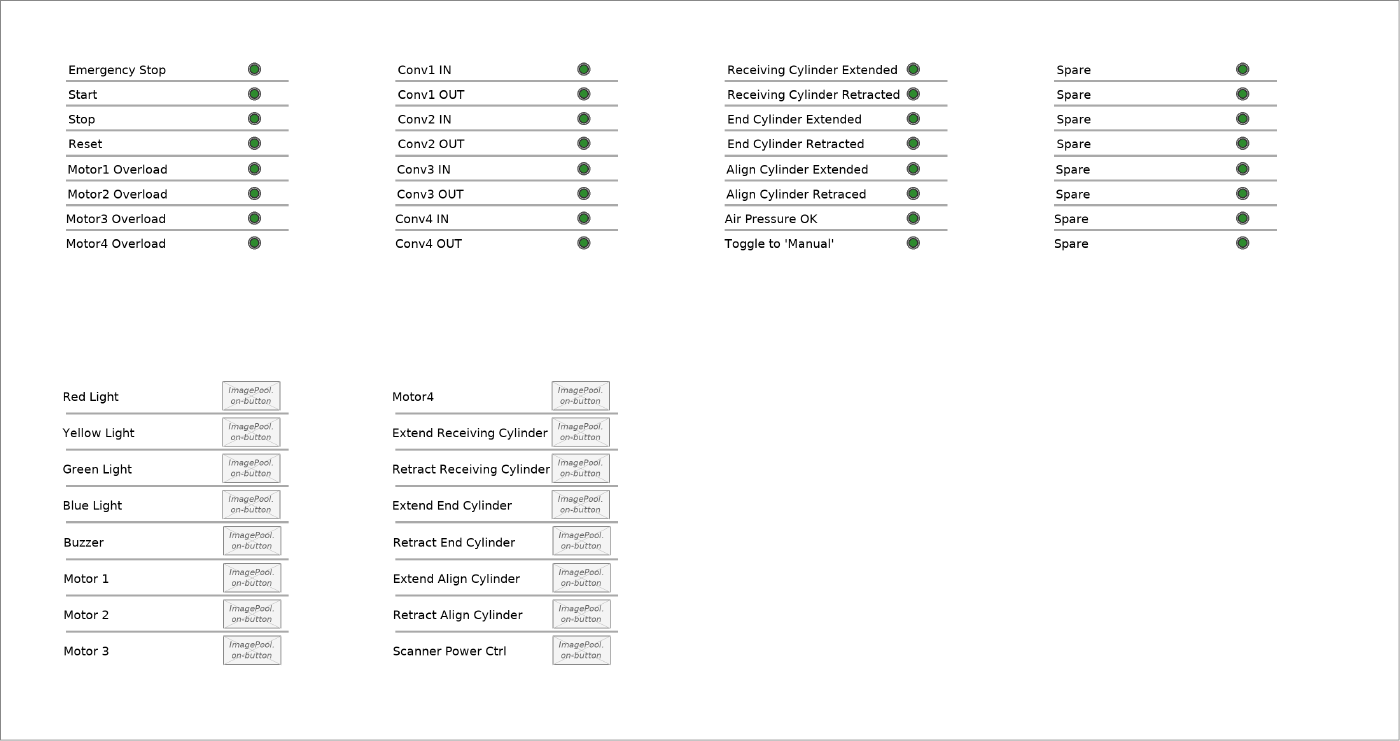
VISUALIZATION PLC_IO_CONTENT  // 1700x900
    Rectangle (0,0 1700x900)
    Group (50,60 300x260)
        RoundedRectangle (0,0 300x260)
        Rectangle (30,10 125x30), "Emergency Stop"
        Rectangle (30,40 118x30), "Start"
        Rectangle (30,70 118x30), "Stop"
        Rectangle (30,100 118x30), "Reset"
        Lamp1 (250,15 18x18), variable: IO_control.bEstop, style: Lamp-Lamp1-Green
        Lamp1 (250,45 18x18), variable: IO_control.bStart, style: Lamp-Lamp1-Green
        Lamp1 (250,75 18x18), variable: IO_control.bStop, style: Lamp-Lamp1-Green
        Lamp1 (250,105 18x18), variable: io_control.bReset, style: Lamp-Lamp1-Green
        Rectangle (30,37 270x2)
        Rectangle (30,67 270x2)
        Rectangle (30,97 270x2)
        Rectangle (29,131 130x30), "Motor1 Overload"
        Rectangle (29,161 200x30), "Motor2 Overload"
        Lamp1 (250,136 18x18), variable: IO.bOverload1, style: Lamp-Lamp1-Green
        Lamp1 (250,166 18x18), variable: IO.bOverload2, style: Lamp-Lamp1-Green
        Rectangle (30,158 270x2)
        Rectangle (30,128 270x2)
        Rectangle (27,191 140x30), "Motor3 Overload"
        Rectangle (27,221 140x30), "Motor4 Overload"
        Lamp1 (250,196 18x18), variable: IO.bOverload3, style: Lamp-Lamp1-Green
        Lamp1 (250,226 18x18), variable: IO.bOverload4, style: Lamp-Lamp1-Green
        Rectangle (30,218 270x2)
        Rectangle (30,188 270x2)
    Group (450,60 300x260)
        RoundedRectangle (0,0 300x260)
        Rectangle (30,10 125x30), "Conv1 IN"
        Rectangle (30,40 125x30), "Conv1 OUT"
        Rectangle (30,70 118x30), "Conv2 IN"
        Rectangle (30,100 118x30), "Conv2 OUT"
        Lamp1 (250,15 18x18), variable: IO.bConv1_In, style: Lamp-Lamp1-Green
        Lamp1 (250,45 18x18), variable: IO.bConv1_Out, style: Lamp-Lamp1-Green
        Lamp1 (250,75 18x18), variable: IO.bConv2_In, style: Lamp-Lamp1-Green
        Lamp1 (250,105 18x18), variable: IO.bConv2_Out, style: Lamp-Lamp1-Green
        Rectangle (30,37 270x2)
        Rectangle (30,67 270x2)
        Rectangle (30,97 270x2)
        Rectangle (29,131 118x30), "Conv3 IN"
        Rectangle (29,161 200x30), "Conv3 OUT"
        Lamp1 (250,136 18x18), variable: IO.bConv3_In, style: Lamp-Lamp1-Green
        Lamp1 (250,166 18x18), variable: IO.bConv3_Out, style: Lamp-Lamp1-Green
        Rectangle (30,158 270x2)
        Rectangle (30,128 270x2)
        Rectangle (27,191 140x30), "Conv4 IN"
        Rectangle (27,221 140x30), "Conv4 OUT"
        Lamp1 (250,196 18x18), variable: IO.bConv4_In, style: Lamp-Lamp1-Green
        Lamp1 (250,226 18x18), variable: IO.bConv4_Out, style: Lamp-Lamp1-Green
        Rectangle (30,218 270x2)
        Rectangle (30,188 270x2)
    Group (850,60 300x260)
        RoundedRectangle (0,0 300x260)
        Rectangle (30,10 210x30), "Receiving Cylinder Extended"
        Rectangle (30,40 210x30), "Receiving Cylinder Retracted"
        Rectangle (30,70 200x30), "End Cylinder Extended"
        Rectangle (30,100 200x30), "End Cylinder Retracted"
        Lamp1 (250,15 18x18), variable: IO.bReCyl1_State_Extend, style: Lamp-Lamp1-Green
        Lamp1 (250,45 18x18), variable: IO.bReCyl1_State_Retract, style: Lamp-Lamp1-Green
        Lamp1 (250,75 18x18), variable: IO.bEndCyl1_State_Extend, style: Lamp-Lamp1-Green
        Lamp1 (250,105 18x18), variable: IO.bEndCyl1_State_Retract, style: Lamp-Lamp1-Green
        Rectangle (30,37 270x2)
        Rectangle (30,67 270x2)
        Rectangle (30,97 270x2)
        Rectangle (29,131 200x30), "Align Cylinder Extended"
        Rectangle (29,161 200x30), "Align Cylinder Retraced"
        Lamp1 (250,136 18x18), variable: IO.bAlCyl1_State_Extend, style: Lamp-Lamp1-Green
        Lamp1 (250,166 18x18), variable: IO.bAlCyl1_State_Retract, style: Lamp-Lamp1-Green
        Rectangle (30,158 270x2)
        Rectangle (30,128 270x2)
        Rectangle (27,191 140x30), "Air Pressure OK"
        Rectangle (27,221 140x30), "Toggle to 'Manual'"
        Lamp1 (250,196 18x18), variable: IO.bPressureOK, style: Lamp-Lamp1-Green
        Lamp1 (250,226 18x18), variable: IO.bManualToggle, style: Lamp-Lamp1-Green
        Rectangle (30,218 270x2)
        Rectangle (30,188 270x2)
    Group (1250,60 300x260)
        RoundedRectangle (0,0 300x260)
        Rectangle (30,10 210x30), "Spare"
        Rectangle (30,40 210x30), "Spare"
        Rectangle (30,70 200x30), "Spare"
        Rectangle (30,100 200x30), "Spare"
        Lamp1 (250,15 18x18), style: Lamp-Lamp1-Green
        Lamp1 (250,45 18x18), style: Lamp-Lamp1-Green
        Lamp1 (250,75 18x18), style: Lamp-Lamp1-Green
        Lamp1 (250,105 18x18), style: Lamp-Lamp1-Green
        Rectangle (30,37 270x2)
        Rectangle (30,67 270x2)
        Rectangle (30,97 270x2)
        Rectangle (29,131 200x30), "Spare"
        Rectangle (29,161 200x30), "Spare"
        Lamp1 (250,136 18x18), style: Lamp-Lamp1-Green
        Lamp1 (250,166 18x18), style: Lamp-Lamp1-Green
        Rectangle (30,158 270x2)
        Rectangle (30,128 270x2)
        Rectangle (27,191 140x30), "Spare"
        Rectangle (27,221 140x30), "Spare"
        Lamp1 (250,196 18x18), style: Lamp-Lamp1-Green
        Lamp1 (250,226 18x18), style: Lamp-Lamp1-Green
        Rectangle (30,218 270x2)
        Rectangle (30,188 270x2)
    Group (50,452 300x366)
        RoundedRectangle (0,0 300x366)
        RoundedRectangle (23,21 109x18), "Red Light"
        RoundedRectangle (23,65 92x18), "Yellow Light"
        RoundedRectangle (23,109 92x18), "Green Light"
        RoundedRectangle (23,153 92x18), "Blue Light"
        Rectangle (30,49 270x2)
        Rectangle (30,93 270x2)
        Rectangle (30,137 270x2)
        RoundedRectangle (24,198 92x18), "Buzzer"
        Rectangle (30,181 270x2)
        RoundedRectangle (24,242 92x18), "Motor 1"
        Rectangle (30,226 270x2)
        RoundedRectangle (24,286 92x18), "Motor 2"
        Rectangle (30,270 270x2)
        RoundedRectangle (24,330 60x18), "Motor 3"
        Image (220,11 70x35), invisible if: IO.bRedLight, image: ImagePool.off-button
            OnMouseClick: toggle IO_HMI.bRedlight
        Image (220,11 70x35), invisible if: NOT IO.bRedLight, image: ImagePool.on-button
            OnMouseClick: toggle IO_HMI.bRedlight
        Image (220,55 70x35), invisible if: IO.bYellowLight, image: ImagePool.off-button
            OnMouseClick: toggle IO_HMI.bYellowlight
        Image (220,55 70x35), invisible if: NOT IO.bYellowLight, image: ImagePool.on-button
            OnMouseClick: toggle IO_HMI.bYellowlight
        Image (220,99 70x35), invisible if: IO.bGreenLight, image: ImagePool.off-button
            OnMouseClick: toggle IO_HMI.bGreenlight
        Image (220,99 70x35), invisible if: NOT IO.bGreenLight, image: ImagePool.on-button
            OnMouseClick: toggle IO_HMI.bGreenlight
        Image (220,143 70x35), image: ImagePool.off-button
            OnMouseClick: toggle 
        Image (220,143 70x35), image: ImagePool.on-button
            OnMouseClick: toggle 
        Image (221,187 70x35), invisible if: IO.bBuzzer, image: ImagePool.off-button
            OnMouseClick: toggle IO_HMI.bBuzzer
        Image (221,187 70x35), invisible if: NOT IO.bBuzzer, image: ImagePool.on-button
            OnMouseClick: toggle IO_HMI.bBuzzer
        Image (221,232 70x35), invisible if: IO.bMotor1, image: ImagePool.off-button
            OnMouseClick: toggle IO_HMI.bMotor1
        Image (221,232 70x35), invisible if: NOT IO.bMotor1, image: ImagePool.on-button
            OnMouseClick: toggle IO_HMI.bMotor1
        Image (221,276 70x35), invisible if: IO.bMotor2, image: ImagePool.off-button
            OnMouseClick: toggle IO_HMI.bMotor2
        Image (221,276 70x35), invisible if: NOT IO.bMotor2, image: ImagePool.on-button
            OnMouseClick: toggle IO_HMI.bMotor2
        Image (221,320 70x35), invisible if: IO.bMotor3, image: ImagePool.off-button
            OnMouseClick: toggle IO_HMI.bMotor3
        Image (221,320 70x35), invisible if: NOT IO.bMotor3, image: ImagePool.on-button
            OnMouseClick: toggle IO_HMI.bMotor3
        Rectangle (30,314 270x2)
    Group (450,452 300x366)
        RoundedRectangle (0,0 300x366)
        RoundedRectangle (23,21 109x18), "Motor4"
        RoundedRectangle (23,65 200x18), "Extend Receiving Cylinder"
        RoundedRectangle (23,109 200x18), "Retract Receiving Cylinder"
        RoundedRectangle (23,153 180x18), "Extend End Cylinder"
        Rectangle (30,49 270x2)
        Rectangle (30,93 270x2)
        Rectangle (30,137 270x2)
        RoundedRectangle (24,198 185x18), "Retract End Cylinder"
        Rectangle (30,181 270x2)
        RoundedRectangle (24,242 180x18), "Extend Align Cylinder"
        Rectangle (30,226 270x2)
        RoundedRectangle (24,286 180x18), "Retract Align Cylinder"
        Rectangle (30,270 270x2)
        RoundedRectangle (24,330 180x18), "Scanner Power Ctrl"
        Image (220,11 70x35), invisible if: IO.bMotor4, image: ImagePool.off-button
            OnMouseClick: toggle IO_HMI.bMotor4
        Image (220,11 70x35), invisible if: NOT IO.bMotor4, image: ImagePool.on-button
            OnMouseClick: toggle IO_HMI.bMotor4
        Image (220,55 70x35), invisible if: IO.bReCyl_Ext, image: ImagePool.off-button
            OnMouseClick: toggle IO_HMI.bRecyl_ext
        Image (220,55 70x35), invisible if: NOT IO.bReCyl_Ext, image: ImagePool.on-button
            OnMouseClick: toggle IO_HMI.bRecyl_ext
        Image (220,99 70x35), invisible if: IO.bReCyl_Ret, image: ImagePool.off-button
            OnMouseClick: toggle IO_HMI.bRecyl_ret
        Image (220,99 70x35), invisible if: NOT IO.bReCyl_Ret, image: ImagePool.on-button
            OnMouseClick: toggle IO_HMI.bRecyl_ret
        Image (220,143 70x35), invisible if: IO.bEndCyl_Ext, image: ImagePool.off-button
            OnMouseClick: toggle IO_HMI.bEndcyl_ext
        Image (220,143 70x35), invisible if: NOT IO.bEndCyl_Ext, image: ImagePool.on-button
            OnMouseClick: toggle IO_HMI.bEndcyl_ext
        Image (221,187 70x35), invisible if: IO.bEndCyl_Ret, image: ImagePool.off-button
            OnMouseClick: toggle IO_HMI.bEndcyl_ret
        Image (221,187 70x35), invisible if: NOT IO.bEndCyl_Ret, image: ImagePool.on-button
            OnMouseClick: toggle IO_HMI.bEndcyl_ret
        Image (221,232 70x35), invisible if: IO.bAlCyl_Ext, image: ImagePool.off-button
            OnMouseClick: toggle IO_HMI.bAlcyl_ext
        Image (221,232 70x35), invisible if: NOT IO.bAlCyl_Ext, image: ImagePool.on-button
            OnMouseClick: toggle IO_HMI.bAlcyl_ext
        Image (221,276 70x35), invisible if: IO.bAlCyl_Ret, image: ImagePool.off-button
            OnMouseClick: toggle IO_HMI.bAlcyl_ret
        Image (221,276 70x35), invisible if: NOT IO.bAlCyl_Ret, image: ImagePool.on-button
            OnMouseClick: toggle IO_HMI.bAlcyl_ret
        Image (221,320 70x35), invisible if: IO.bScanner_PowerState, image: ImagePool.off-button
            OnMouseClick: toggle IO_HMI.bScanner_PwrCtrl
        Image (221,320 70x35), invisible if: NOT IO.bScanner_PowerState, image: ImagePool.on-button
            OnMouseClick: toggle IO_HMI.bScanner_PwrCtrl
        Rectangle (30,314 270x2)
END_VISUALIZATION

(* stored: Version 1.1.0.1, ProductVersion 3.1.4024.12
   Visu PLC_IO_CONTENT: Id {e8cee26a-39ef-4cf2-901c-7210f9b1a9cd} *)
